FUNCTION_BLOCK fbValueOutOfRange
VAR_INPUT
	r_Min				:REAL;
	r_Max				:REAL;
	r_WhenError			:REAL;
END_VAR

VAR_IN_OUT
	r_var				:REAL;
END_VAR

VAR_OUTPUT
	Q					:BOOL;
	r_Out				:REAL;	
	b_IsError			:BOOL;
END_VAR

IF r_var >= r_Min AND r_var <= r_Max THEN
	Q := TRUE;
ELSE
	Q := FALSE;
	r_var := r_WhenError;
END_IF

b_IsError := NOT Q;
r_Out := r_var;

END_FUNCTION_BLOCK

(* stored: Version 1.1.0.1, ProductVersion 3.1.4026.18
   POU fbValueOutOfRange: Id {624ae231-1f9f-4297-8486-4ea2685772f9}, SpecialFunc None *)
